FUNCTION_BLOCK FB_Observable_WORD EXTENDS FB_AbstractObservable
VAR
    _nVal:              WORD;
    _nOldVal:           WORD;
END_VAR

METHOD FB_init : BOOL
VAR_INPUT
    bInitRetains:       BOOL; // if TRUE, the retain variables are initialized (warm start / cold start)
    bInCopyCode:        BOOL;  // if TRUE, the instance afterwards gets moved into the copy code (online change)
END_VAR
THIS^._nTypeClass := __SYSTEM.TYPE_CLASS.TYPE_WORD;
END_METHOD

PROPERTY nDataSize : UDINT
GET
nDataSize := SIZEOF(WORD);
END_GET
END_PROPERTY

PROPERTY nValue16 : WORD
GET
nValue16 := THIS^._nVal;
END_GET
SET
THIS^._nOldVal := THIS^._nVal;
THIS^._nVal := nValue16;

THIS^.NotifyWithConditions();
END_SET
END_PROPERTY

PROPERTY PROTECTED pData : POINTER TO BYTE
GET
pData := ADR(THIS^._nVal);
END_GET
END_PROPERTY

METHOD  ValueChanged : BOOL
VAR_INPUT
END_VAR
ValueChanged := THIS^._nOldVal <> THIS^._nVal;
END_METHOD

END_FUNCTION_BLOCK

(* stored: Version 1.1.0.1, ProductVersion 3.1.4024.12
   POU FB_Observable_WORD: Id {ebc0a468-fb5d-0457-1f66-b1daed1d4150}, SpecialFunc None
   Method FB_init: Id {4fa35d8c-175e-09c3-1fac-7d470c2ce0df}
   Property nDataSize: Id {f2ff5b99-b352-0410-2d16-7ee056f2c4c9}
   Get Get: Id {032c87eb-6b15-0906-175c-2a814ad1222e}
   Property nValue16: Id {5e13c9b8-4784-0cd7-3a89-6406ca1952a8}
   Get Get: Id {18ba444b-ed87-0508-3604-030fdb51b5db}
   Set Set: Id {da68199d-cb5c-095d-0375-99e2c4d09c42}
   Property pData: Id {5c1b2ca7-ad37-0472-136c-7b522c896b88}
   Get Get: Id {99162a72-4d46-09da-0df7-82dcc90a57ab}
   Method ValueChanged: Id {c574f09d-b78d-0449-03bd-3423bdfb3be3} *)
